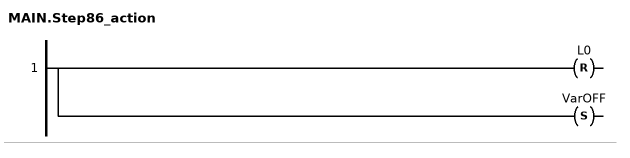
[picture p24: MAIN.Step86_action (LD)]
_LD_ (* Ladder Diagram *)
NETWORK 1
	* --- (R L0) (S VarOFF)
_END_LD_
(* the same logic as Structured Text *)
(* Network 1 *)
L0 := FALSE;
VarOFF := TRUE;
END_ACTION

ACTION Rot1pt2_action:
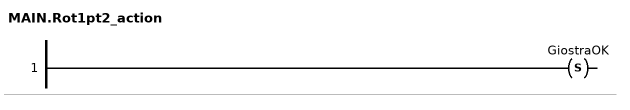
_LD_ (* Ladder Diagram *)
NETWORK 1
	* --- (S GiostraOK)
_END_LD_
(* the same logic as Structured Text *)
(* Network 1 *)
GiostraOK := TRUE;
END_ACTION

ACTION Step782_action:
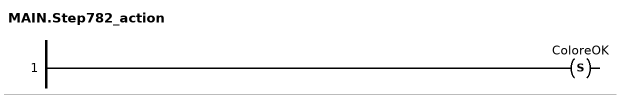
_LD_ (* Ladder Diagram *)
NETWORK 1
	* --- (S ColoreOK)
_END_LD_
(* the same logic as Structured Text *)
(* Network 1 *)
ColoreOK := TRUE;
END_ACTION

ACTION Rot1_action:
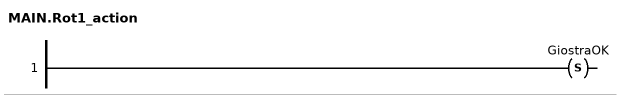
_LD_ (* Ladder Diagram *)
NETWORK 1
	* --- (S GiostraOK)
_END_LD_
(* the same logic as Structured Text *)
(* Network 1 *)
GiostraOK := TRUE;
END_ACTION

ACTION Step78_action:
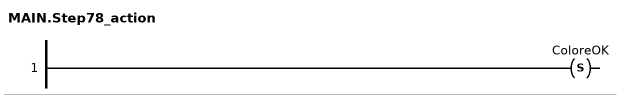
_LD_ (* Ladder Diagram *)
NETWORK 1
	* --- (S ColoreOK)
_END_LD_
(* the same logic as Structured Text *)
(* Network 1 *)
ColoreOK := TRUE;
END_ACTION

ACTION Rotazione_action:
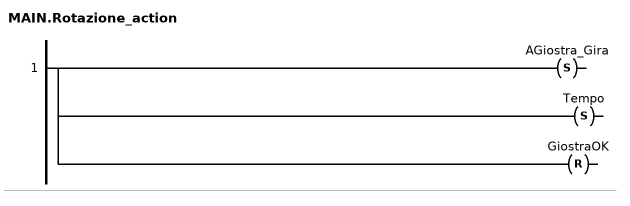
_LD_ (* Ladder Diagram *)
NETWORK 1
	* --- (S AGiostra_Gira) (S Tempo) (R GiostraOK)
_END_LD_
(* the same logic as Structured Text *)
(* Network 1 *)
AGiostra_Gira := TRUE;
Tempo := TRUE;
GiostraOK := FALSE;
END_ACTION

ACTION ResetGiostra_action:
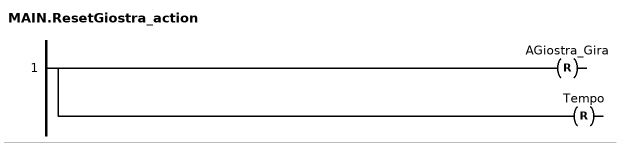
_LD_ (* Ladder Diagram *)
NETWORK 1
	* --- (R AGiostra_Gira) (R Tempo)
_END_LD_
(* the same logic as Structured Text *)
(* Network 1 *)
AGiostra_Gira := FALSE;
Tempo := FALSE;
END_ACTION

ACTION ResetColore_action:
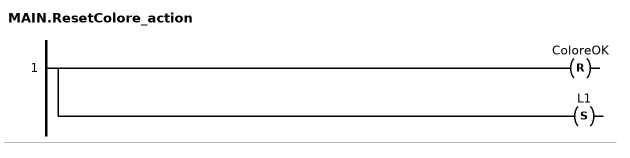
_LD_ (* Ladder Diagram *)
NETWORK 1
	* --- (R ColoreOK) (S L1)
_END_LD_
(* the same logic as Structured Text *)
(* Network 1 *)
ColoreOK := FALSE;
L1 := TRUE;
END_ACTION

ACTION SetRed_action:
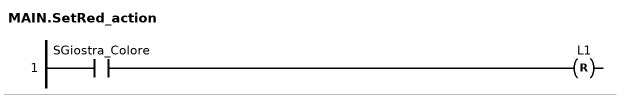
_LD_ (* Ladder Diagram *)
NETWORK 1
	[SGiostra_Colore] --- (R L1)
_END_LD_
(* the same logic as Structured Text *)
(* Network 1 *)
IF SGiostra_Colore THEN L1 := FALSE; END_IF;
END_ACTION

ACTION Rot2_action:
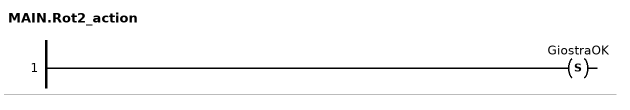
_LD_ (* Ladder Diagram *)
NETWORK 1
	* --- (S GiostraOK)
_END_LD_
(* the same logic as Structured Text *)
(* Network 1 *)
GiostraOK := TRUE;
END_ACTION

ACTION Step788_action:
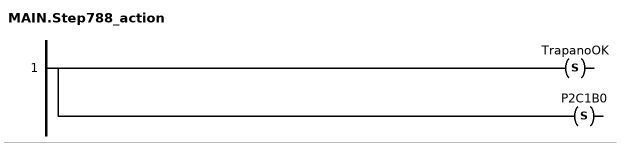
_LD_ (* Ladder Diagram *)
NETWORK 1
	* --- (S TrapanoOK) (S P2C1B0)
_END_LD_
(* the same logic as Structured Text *)
(* Network 1 *)
TrapanoOK := TRUE;
P2C1B0 := TRUE;
END_ACTION

ACTION SetNotRed_action:
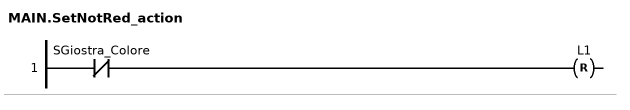
_LD_ (* Ladder Diagram *)
NETWORK 1
	[/SGiostra_Colore] --- (R L1)
_END_LD_
(* the same logic as Structured Text *)
(* Network 1 *)
IF NOT SGiostra_Colore THEN L1 := FALSE; END_IF;
END_ACTION

ACTION Rot3_action:
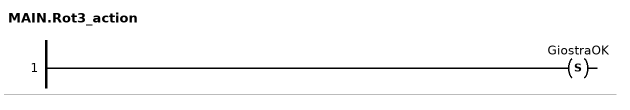
_LD_ (* Ladder Diagram *)
NETWORK 1
	* --- (S GiostraOK)
_END_LD_
(* the same logic as Structured Text *)
(* Network 1 *)
GiostraOK := TRUE;
END_ACTION

ACTION Step799_action:
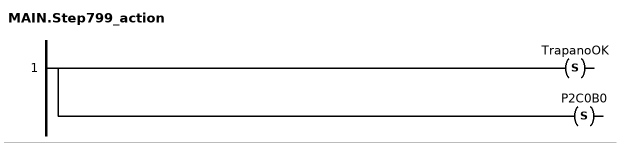
_LD_ (* Ladder Diagram *)
NETWORK 1
	* --- (S TrapanoOK) (S P2C0B0)
_END_LD_
(* the same logic as Structured Text *)
(* Network 1 *)
TrapanoOK := TRUE;
P2C0B0 := TRUE;
END_ACTION

ACTION ResetTrapano_action:
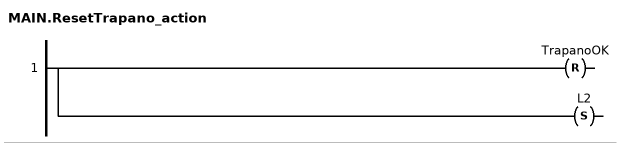
_LD_ (* Ladder Diagram *)
NETWORK 1
	* --- (R TrapanoOK) (S L2)
_END_LD_
(* the same logic as Structured Text *)
(* Network 1 *)
TrapanoOK := FALSE;
L2 := TRUE;
END_ACTION

ACTION Fora_action:
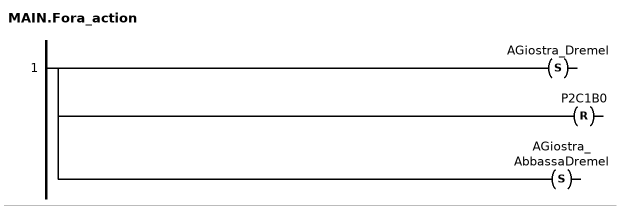
_LD_ (* Ladder Diagram *)
NETWORK 1
	* --- (S AGiostra_Dremel) (R P2C1B0) (S AGiostra_AbbassaDremel)
_END_LD_
(* the same logic as Structured Text *)
(* Network 1 *)
AGiostra_Dremel := TRUE;
P2C1B0 := FALSE;
AGiostra_AbbassaDremel := TRUE;
END_ACTION

ACTION RitornoTrapano_action:
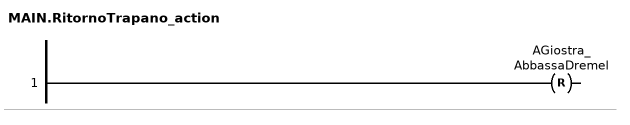
_LD_ (* Ladder Diagram *)
NETWORK 1
	* --- (R AGiostra_AbbassaDremel)
_END_LD_
(* the same logic as Structured Text *)
(* Network 1 *)
AGiostra_AbbassaDremel := FALSE;
END_ACTION

ACTION Spegni_action:
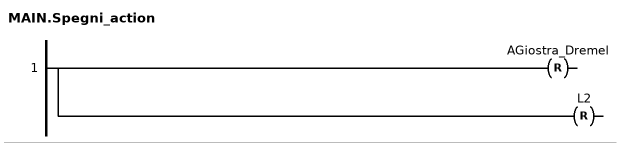
_LD_ (* Ladder Diagram *)
NETWORK 1
	* --- (R AGiostra_Dremel) (R L2)
_END_LD_
(* the same logic as Structured Text *)
(* Network 1 *)
AGiostra_Dremel := FALSE;
L2 := FALSE;
END_ACTION

ACTION Rot4_action:
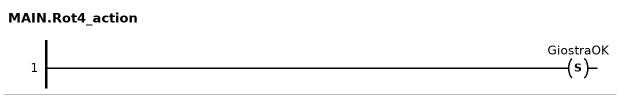
_LD_ (* Ladder Diagram *)
NETWORK 1
	* --- (S GiostraOK)
_END_LD_
(* the same logic as Structured Text *)
(* Network 1 *)
GiostraOK := TRUE;
END_ACTION

ACTION Step102_action:
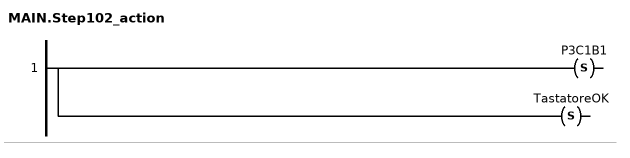
_LD_ (* Ladder Diagram *)
NETWORK 1
	* --- (S P3C1B1) (S TastatoreOK)
_END_LD_
(* the same logic as Structured Text *)
(* Network 1 *)
P3C1B1 := TRUE;
TastatoreOK := TRUE;
END_ACTION

ACTION SetVar_action:
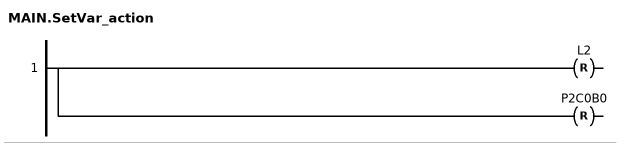
_LD_ (* Ladder Diagram *)
NETWORK 1
	* --- (R L2) (R P2C0B0)
_END_LD_
(* the same logic as Structured Text *)
(* Network 1 *)
L2 := FALSE;
P2C0B0 := FALSE;
END_ACTION

ACTION Rot5_action:
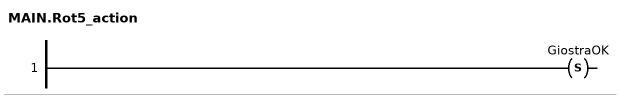
_LD_ (* Ladder Diagram *)
NETWORK 1
	* --- (S GiostraOK)
_END_LD_
(* the same logic as Structured Text *)
(* Network 1 *)
GiostraOK := TRUE;
END_ACTION

ACTION Step101_action:
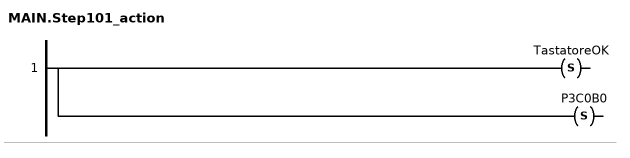
_LD_ (* Ladder Diagram *)
NETWORK 1
	* --- (S TastatoreOK) (S P3C0B0)
_END_LD_
(* the same logic as Structured Text *)
(* Network 1 *)
TastatoreOK := TRUE;
P3C0B0 := TRUE;
END_ACTION

ACTION ResetTastatore_action:
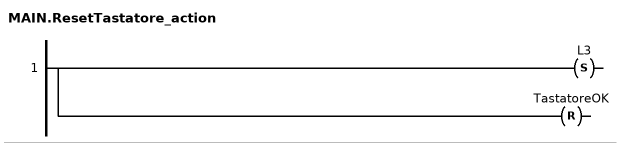
_LD_ (* Ladder Diagram *)
NETWORK 1
	* --- (S L3) (R TastatoreOK)
_END_LD_
(* the same logic as Structured Text *)
(* Network 1 *)
L3 := TRUE;
TastatoreOK := FALSE;
END_ACTION

ACTION AbbassaTastatore_action:
